FUNCTION_BLOCK FB_ReadTextFromFile
VAR_INPUT
	bExecute		: BOOL;			(* Komenda odczytu *)
	AmsNetId		: T_AmsNetId;	(* AMS NET ID obiektu docelowego, gdy lokalnie, to zmienna moze byc pusta *)
	sPath			: STRING; 		(* Sciezka pliku, np  'Hard Disk\'*)
	sName			: STRING; 		(* Nazwa pliku wraz z rozszerzeniem 'LogFile.txt'; *)
END_VAR

VAR_OUTPUT
	bBusy		: BOOL;
	bError		: BOOL;
	sLine		: STRING;		(* Tresc wpisu *)
END_VAR
VAR
	fbFileOpen	: FB_FileOpen;
	ftOpen		: F_TRIG;
	fbFileGets	: FB_FileGets;
	ftGets		: F_TRIG;
	fbFileClose	: FB_FileClose;
	ftClose		: F_TRIG;
END_VAR
VAR // added by the converter: edge detectors and wires of the graphical bodies
    _w1 : BOOL;
END_VAR

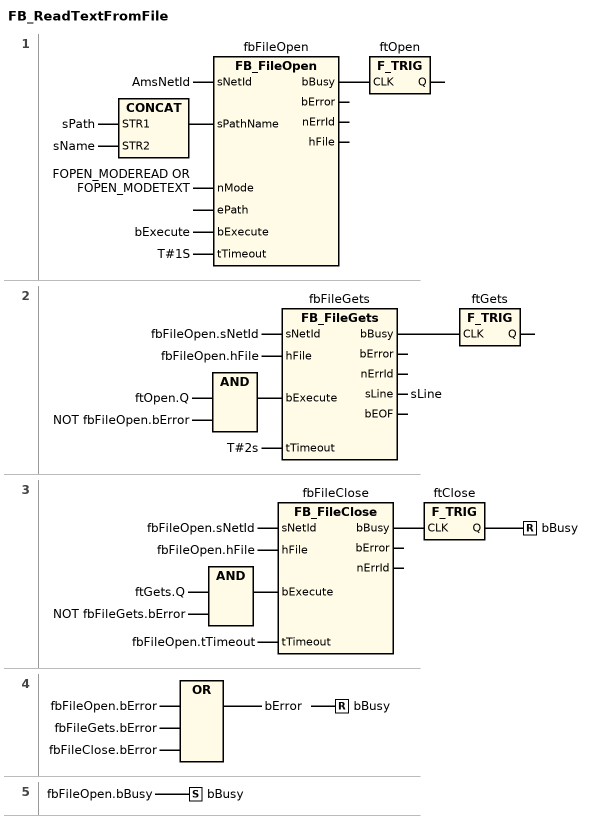
// NETWORK 1
fbFileOpen(
    sNetId := AmsNetId,
    sPathName := CONCAT(STR1 := sPath, STR2 := sName),
    nMode := FOPEN_MODEREAD OR FOPEN_MODETEXT,
    bExecute := bExecute,
    tTimeout := T#1S); // FB_FileOpen
ftOpen(CLK := fbFileOpen.bBusy); // F_TRIG

// NETWORK 2
fbFileGets(
    sNetId := fbFileOpen.sNetId,
    hFile := fbFileOpen.hFile,
    bExecute := ftOpen.Q AND (NOT fbFileOpen.bError),
    tTimeout := T#2s,
    sLine => sLine); // FB_FileGets
ftGets(CLK := fbFileGets.bBusy); // F_TRIG

// NETWORK 3
fbFileClose(
    sNetId := fbFileOpen.sNetId,
    hFile := fbFileOpen.hFile,
    bExecute := ftGets.Q AND (NOT fbFileGets.bError),
    tTimeout := fbFileOpen.tTimeout); // FB_FileClose
ftClose(CLK := fbFileClose.bBusy); // F_TRIG
bBusy R= ftClose.Q;

// NETWORK 4
_w1 := fbFileOpen.bError OR fbFileGets.bError OR fbFileClose.bError;
bError := _w1;
bBusy R= _w1;

// NETWORK 5
bBusy S= fbFileOpen.bBusy;

END_FUNCTION_BLOCK

(* stored: Version 1.1.0.1, ProductVersion 3.1.4026.13, FileIdentifier ffb8dc3902ece8a7756dad997a30d9ee66cd623b, FileSignature 655f6360e9efc1bee78f1d3a60a84a6dc1e20c7b15406f0eefe7c485c1723a86308befc87e647d96871571aa02f016f5e6649c82ac43c175d97613560e937d445664548284d63ad1de3687857c298c9ccca63397d99914cf52625007082f894558285d424ab2c87e89918e570029c050577acfc7ac8675e7cc431354c959a0c39a095c1cfc5088eacb7fd3e1e35acf042696d17eb900d5d4e42b1462fc8de81cfc9c05a13042a231b18581e7a3d60893f0a64b93378544995f3834898caa5a0ae197622559c5520a9da1a42ed958d6b04042e5b5bb12be9f494723b936f307fb5bfc87d47d1847deeae8bb9fc370e894ec34c8646e831254eb773718b6f712ad
   POU FB_ReadTextFromFile: Id {4b7c7c9a-b915-4045-a02f-3004e6b0f94f}, SpecialFunc None *)
